FUNCTION_BLOCK FBBTN
VAR_INPUT
	bOLD : BOOL;
	bNEW : BOOL;
END_VAR
VAR_OUTPUT
	bOUT : BOOL;
END_VAR
VAR
END_VAR

IF bOLD = FALSE AND bNEW = TRUE THEN
	bOUT := TRUE;
ELSE
	bOUT := FALSE;
END_IF

bOLD := bNEW;

END_FUNCTION_BLOCK

(* stored: Version 1.1.0.1, ProductVersion 3.1.4026.18
   POU FBBTN: Id {40759bd4-0b0b-44b1-82ac-fd9964b597b6}, SpecialFunc None *)
